Yaskawa INFORM job: MASTER_X2.JBI

/JOB
//NAME MASTER_X2
///FOLDERNAME MASTER_ODWLOK
//POS
///NPOS 131,131,131,0,0,0
///TOOL 0
///POSTYPE PULSE
///PULSE
C00000=-2000,-113621,-91819,0,89172,0
C00001=-2000,-113621,-91819,0,89172,0
C00002=-2032,-101495,-83135,17,53290,-13
C00003=-2000,-48025,-60869,0,102856,0
C00004=-3643,-76224,-106676,-19950,71810,-76872
C00005=-3643,-76224,-106676,-19950,71810,-76872
C00006=-2000,-130321,-133031,0,28968,0
C00007=-2000,-109649,-128472,0,44436,0
C00008=-2000,-75195,-120874,0,70216,0
C00009=-2000,-52226,-115808,0,87402,0
C00010=-2000,-87067,-95572,0,78525,0
C00011=-2000,-87067,-95572,0,78525,0
C00012=-2000,-87067,-95572,0,78525,0
C00013=12667,-135547,-130714,-31270,45596,0
C00014=12667,-135547,-130714,-31270,45596,0
C00015=12667,-135547,-130714,-31270,45596,0
C00016=7337,-135032,-132177,-15524,30149,-37578
C00017=1415,-134459,-133802,1969,12985,-79332
C00018=1415,-134459,-133802,1969,12985,-79332
C00019=15972,-110889,-128286,10965,59905,43045
C00020=-2800,-56338,-97337,367,83074,-232
C00021=-2800,-56338,-97337,367,83074,-232
C00022=-2000,-92772,-84335,0,66375,0
C00023=-2000,-92772,-84335,0,66375,0
C00024=-2000,-92772,-84335,0,66375,0
C00025=-2000,-92772,-84335,0,66375,0
C00026=-2000,-92055,-48789,0,51065,0
C00027=-2000,-92055,-48789,0,51065,0
C00028=-2000,-92055,-48789,0,51065,0
C00029=-2000,-92055,-48789,0,51065,0
C00030=-2348,-136985,-121477,-16,96092,-119
C00031=-2348,-136985,-121477,-16,96092,-119
C00032=-2348,-136985,-121477,-16,96092,-119
C00033=9622,-119744,-117240,-5707,89112,-22022
C00034=39612,-76551,-106625,-19964,71626,-76894
C00035=8691,-94790,-119167,-5108,91578,-19600
C00036=-1903,-101039,-123464,-18,98414,30
C00037=-1903,-101039,-123464,-18,98414,30
C00038=-1903,-101039,-123464,-18,98414,30
C00039=-1903,-101039,-123464,-18,98414,30
C00040=39612,-76551,-106625,-19964,71626,-76894
C00041=39612,-76551,-106625,-19964,71626,-76894
C00042=39612,-76551,-106625,-19964,71626,-76894
C00043=39612,-76551,-106625,-19964,71626,-76894
C00044=39612,-76551,-106625,-19964,71626,-76894
C00045=39612,-76551,-106625,-19964,71626,-76894
C00046=39612,-76551,-106625,-19964,71626,-76894
C00047=39612,-76551,-106625,-19964,71626,-76894
C00048=39612,-76551,-106625,-19964,71626,-76894
C00049=10776,-116726,-133110,-1428,79202,-268
C00050=10776,-116726,-133110,-1428,79202,-268
C00051=10907,-117335,-90652,18762,63715,59495
C00052=10907,-117335,-90652,18762,63715,59495
C00053=10776,-116726,-133110,-1428,79202,-268
C00054=10776,-116726,-133110,-1428,79202,-268
C00055=10907,-117335,-90652,18762,63715,59495
C00056=-2286,-107682,-96534,81,71711,-101
C00057=-2286,-107682,-96534,81,71711,-101
C00058=-2286,-107682,-96534,81,71711,-101
C00059=-2000,-113393,-91320,0,88983,0
C00060=-2000,-113393,-91320,0,88983,0
C00061=-2000,-113393,-91320,0,88983,0
C00062=-2000,-113393,-91320,0,88983,0
C00063=-2000,-113393,-91320,0,88983,0
C00064=39612,-76551,-106625,-19964,71626,-76894
C00065=39612,-76551,-106625,-19964,71626,-76894
C00066=39612,-76551,-106625,-19964,71626,-76894
C00067=39612,-76551,-106625,-19964,71626,-76894
C00068=39612,-76551,-106625,-19964,71626,-76894
C00069=39612,-76551,-106625,-19964,71626,-76894
C00070=-15532,205449,169164,0,-1122,-37
C00071=2435,135546,115697,-1555,71481,-4054
C00072=2435,135546,115697,-1555,71481,-4054
C00073=-5072,204191,173913,2520,2133,2072
C00074=-5072,204191,173913,2520,52116,2072
C00075=-3643,-76224,-106676,-19950,71810,-76872
C00076=-1588,-95931,-85547,536,91020,79
C00077=-1588,-95931,-85547,536,91020,79
C00078=-2000,-138093,-117084,0,0,0
C00079=-3643,-76224,-106676,-19950,71810,-76872
C00080=-2000,-138093,-117084,0,0,0
C00081=-2000,-138093,-117084,0,0,0
C00082=-1941,-102693,-129564,-10,101994,18
C00083=-3643,-76224,-106676,-19950,71810,-76872
C00084=-1074,-84890,-111921,-820,92639,133
C00085=-1074,-84890,-111921,-820,92639,133
C00086=-1999,-107637,-123410,0,80759,-1
C00087=-3643,-76224,-106676,-19950,71810,-76872
C00088=-2000,17994,-60377,0,102988,0
C00089=-2000,-95440,-72516,0,38121,0
C00090=-1074,-84890,-111921,-820,92639,133
C00091=-3643,-76224,-106676,-19950,71810,-76872
C00092=-421,-73083,-90384,286,80877,488
C00093=-421,-73083,-90384,286,80877,488
C00094=-2000,-112988,-119327,0,83158,0
C00095=-3643,-76224,-106676,-19950,71810,-76872
C00096=-2000,-112988,-119327,0,83158,0
C00097=-2000,-112988,-119327,0,83158,0
C00098=-2000,-112988,-119327,0,83158,0
C00099=-2000,-112988,-119327,0,83158,0
C00100=-2082,-130750,-111396,32,62200,-31
C00101=-3643,-76224,-106676,-19950,71810,-76872
C00102=-2082,-130750,-111396,32,62200,-31
C00103=-2082,-130750,-111396,32,62200,-31
C00104=-1579,-114561,-88072,-141,60969,160
C00105=-1579,-114561,-88072,-141,60969,160
C00106=-1579,-114561,-88072,-141,60969,160
C00107=-3643,-76224,-106676,-19950,71810,-76872
C00108=137109,-187493,-133090,-6705,82774,76786
C00109=-3643,-76224,-106676,-19950,71810,-76872
C00110=-1579,-114561,-88072,-141,60969,160
C00111=-2027,-78555,-65913,-1,89981,-9
C00112=-3643,-76224,-106676,-19950,71810,-76872
C00113=-2027,-78555,-65913,-1,89981,-9
C00114=-2027,-78555,-65913,-1,89981,-9
C00115=-3322,-122452,-100913,73,83322,-449
C00116=-3643,-76224,-106676,-19950,71810,-76872
C00117=-3322,-122452,-100913,73,83322,-449
C00118=-3322,-122452,-100913,73,83322,-449
C00119=-3322,-122452,-100913,73,83322,-449
C00120=-3322,-122452,-100913,73,83322,-449
C00121=-3322,-122452,-100913,73,83322,-449
C00122=-2847,-120416,-115970,194,80716,-285
C00123=-2000,-115920,-83969,0,54247,0
C00124=-2000,-115920,-83969,0,54247,0
C00125=-3271,-119374,-120746,350,28955,-423
C00126=-3271,-119374,-120746,350,28955,-423
C00127=-3270,-119374,-120745,350,28960,-423
C00128=-3270,-119374,-120745,350,28960,-423
C00129=-3271,-119374,-120746,350,28955,-423
C00130=-2000,-115588,-91819,0,89172,0
BC00000=87173,519039,860034
BC00001=87173,500620,1075193
BC00002=1577,523905,302382
BC00003=118448,523905,678960
BC00004=199448,515539,1075137
BC00005=199448,515539,1075137
BC00006=200118,491577,1075193
BC00007=160304,500134,1054011
BC00008=93948,514396,1018707
BC00009=49710,523905,995172
BC00010=66564,515818,1075139
BC00011=66564,515818,1075139
BC00012=66564,515818,1075139
BC00013=78377,519142,1075139
BC00014=78377,519142,1075139
BC00015=78377,519142,1075139
BC00016=64373,510676,1075139
BC00017=48813,501269,1075139
BC00018=48813,501269,1075139
BC00019=21198,517278,1075139
BC00020=194066,523905,1075139
BC00021=194066,523905,1075139
BC00022=244938,523905,1064782
BC00023=244938,523905,1063114
BC00024=244938,523905,804554
BC00025=244938,523905,1062363
BC00026=198867,523905,1060460
BC00027=198867,523905,1063860
BC00028=198867,523905,632202
BC00029=198867,523905,632202
BC00030=133244,518772,1075139
BC00031=133244,518772,1075139
BC00032=133244,518772,1075139
BC00033=179478,517852,1075139
BC00034=295309,515546,1075139
BC00035=207944,518721,1071325
BC00036=178010,519809,1070018
BC00037=178010,519809,1070018
BC00038=178010,519809,1070018
BC00039=178010,519809,1070018
BC00040=295309,515546,1075139
BC00041=295309,515546,1075139
BC00042=295309,515546,1075139
BC00043=295309,515546,1075139
BC00044=295309,515546,1075139
BC00045=295309,515546,1075139
BC00046=295309,515546,1075139
BC00047=295309,515546,1075139
BC00048=295309,515546,1075139
BC00049=165804,522273,1075193
BC00050=165804,522273,1075193
BC00051=165804,522273,534000
BC00052=165804,608579,806934
BC00053=165804,522273,1075193
BC00054=165804,522273,1075193
BC00055=165804,522273,534000
BC00056=84290,518606,1075193
BC00057=84290,518606,1075193
BC00058=84290,518606,1075193
BC00059=87173,523905,1075193
BC00060=87173,523905,1075193
BC00061=87173,523905,1075193
BC00062=87173,523905,1075193
BC00063=87173,523905,1075193
BC00064=295309,515546,1075139
BC00065=295309,515546,1075139
BC00066=295309,515546,1075139
BC00067=295309,515546,1075139
BC00068=295309,515546,1075139
BC00069=295309,515546,1075139
BC00070=1577,514581,1075193
BC00071=23362,568996,1042628
BC00072=23362,568996,1042628
BC00073=21044,590463,17935
BC00074=21044,590463,17935
BC00075=199448,582493,1075137
BC00076=197629,523905,680388
BC00077=197629,523905,680388
BC00078=166704,523889,1057027
BC00079=199448,515539,1075137
BC00080=166704,523889,1057027
BC00081=166704,523889,1057027
BC00082=210602,521349,578617
BC00083=199448,515539,1075137
BC00084=166156,519383,387149
BC00085=166156,519383,1064329
BC00086=108222,519829,1065853
BC00087=199448,515539,1075137
BC00088=32574,515576,986534
BC00089=30845,523905,744523
BC00090=166156,519383,1045384
BC00091=199448,515539,1075137
BC00092=146427,523905,652589
BC00093=146427,523905,652589
BC00094=91885,523905,1075139
BC00095=199448,515539,1075137
BC00096=91885,523905,1075139
BC00097=91885,523905,1075139
BC00098=91885,523905,1075139
BC00099=91885,523905,1075139
BC00100=147852,523905,1075139
BC00101=199448,515539,1075137
BC00102=147852,523905,1075139
BC00103=147852,523905,1075139
BC00104=127037,517515,1075193
BC00105=127037,517515,1075193
BC00106=127037,517515,1075193
BC00107=199448,515539,1075137
BC00108=267017,506351,1057956
BC00109=199448,515539,1075137
BC00110=127037,517515,1075193
BC00111=1577,523905,1063536
BC00112=199448,515539,1075137
BC00113=1577,523905,619430
BC00114=1577,523905,619430
BC00115=87745,523889,1075193
BC00116=199448,515539,1075137
BC00117=87745,523889,1075193
BC00118=87745,523889,1075193
BC00119=87745,523889,1075193
BC00120=87745,523889,1075193
BC00121=87745,523889,1075193
BC00122=780,523905,878730
BC00123=262874,523905,990511
BC00124=262874,523905,990511
BC00125=132367,523905,1075193
BC00126=132367,523905,1075193
BC00127=132367,523905,1075190
BC00128=132367,523905,1075190
BC00129=132367,523905,1075193
BC00130=86218,606896,448189
EC00000=0,-183832
EC00001=0,-183832
EC00002=-798156,-183832
EC00003=-798156,-1296783
EC00004=-798156,-1296783
EC00005=-306282,-1296783
EC00006=798156,-1296783
EC00007=869104,-1018545
EC00008=869104,-462069
EC00009=798156,-183832
EC00010=798156,-1296783
EC00011=266052,-1296783
EC00012=-266052,-183832
EC00013=-798156,-183832
EC00014=-798156,-183832
EC00015=-266052,-183832
EC00016=-266052,-740307
EC00017=-266052,-1296783
EC00018=-798156,-1296783
EC00019=-798156,-1296783
EC00020=798156,-183832
EC00021=266052,-183832
EC00022=-266052,-1296783
EC00023=-798156,-1296783
EC00024=-798156,-1296783
EC00025=-266052,-1296783
EC00026=5855,-183832
EC00027=-798156,-183832
EC00028=-798156,-183832
EC00029=-266052,-183832
EC00030=443420,372643
EC00031=798156,372643
EC00032=266052,372643
EC00033=-240191,-131321
EC00034=-1507629,-183832
EC00035=-1445784,372643
EC00036=-1330261,372643
EC00037=-1330261,372643
EC00038=-1596313,372643
EC00039=-1507629,-183832
EC00040=1507629,-183832
EC00041=1596313,372643
EC00042=1463287,372643
EC00043=1463287,372643
EC00044=1463287,372643
EC00045=1463287,372643
EC00046=1596313,372643
EC00047=1596313,-183832
EC00048=266052,-183832
EC00049=-266052,-1296783
EC00050=-798156,-1296783
EC00051=-798156,-1296783
EC00052=-266052,-1296783
EC00053=-266052,-183832
EC00054=-798156,-183832
EC00055=-798156,-183832
EC00056=-798156,-183832
EC00057=-798156,-183832
EC00058=-266052,-183832
EC00059=-266052,-1296783
EC00060=-798156,-1296783
EC00061=-798156,-1296783
EC00062=-266052,-1296783
EC00063=266052,-183832
EC00064=1507629,-183832
EC00065=1596313,372643
EC00066=1463287,372643
EC00067=1463287,372643
EC00068=1596313,372643
EC00069=1507629,-183832
EC00070=266052,-183832
EC00071=-2992,-740304
EC00072=1108548,-740304
EC00073=1108551,-740307
EC00074=1108551,-740307
EC00075=-798155,-740307
EC00076=-798156,-740307
EC00077=-266052,-740307
EC00078=-266052,372643
EC00079=-798156,372643
EC00080=-798156,372643
EC00081=-266052,372643
EC00082=-266052,-183832
EC00083=-798156,-183832
EC00084=-798156,-183832
EC00085=-266052,-183832
EC00086=266050,-1296783
EC00087=798156,-1296783
EC00088=798156,-183832
EC00089=266052,-183832
EC00090=-266052,-1296783
EC00091=-798156,-1296783
EC00092=-798156,-1296783
EC00093=-1596313,-1296783
EC00094=-1596313,372643
EC00095=-1330261,372643
EC00096=-1330261,372643
EC00097=-1596313,372643
EC00098=-1507629,-183832
EC00099=-266052,-183832
EC00100=-266052,-740307
EC00101=-780419,-740307
EC00102=-780419,-740307
EC00103=-266052,-740307
EC00104=266052,-183832
EC00105=798156,-183832
EC00106=1585256,-183832
EC00107=1527674,-741132
EC00108=1488721,-182878
EC00109=798156,-183832
EC00110=-266052,-183832
EC00111=-266052,-740307
EC00112=-798154,-740306
EC00113=-798156,-740307
EC00114=-266052,-740307
EC00115=-266052,-1296783
EC00116=-798156,-1296783
EC00117=-798156,-1296783
EC00118=-266052,-1296783
EC00119=-266052,-183832
EC00120=-798156,-183832
EC00121=-798156,-183832
EC00122=-1596313,-183832
EC00123=-1596313,372643
EC00124=-1596313,-183832
EC00125=-266052,-183832
EC00126=-266052,-740307
EC00127=77843,371283
EC00128=77843,371283
EC00129=0,-183832
EC00130=0,-183832
//INST
///DATE 2024/12/18 17:27
///ATTR SC,RW
///GROUP1 RB1,BS1
///GROUP2 ST1
NOP
WAIT IG#(285)=255
CLEAR B060 1
'MASTER
SETTM TM000 TRESET
SETTM TM000 TSTART
COMM DOUT OT#(1433) ON
DOUT OT#(1437) ON
MOVJ C00000 BC00000 VJ=100.00  +MOVJ EC00000 VJ=100.00
MOVJ C00001 BC00001 VJ=100.00  +MOVJ EC00001 VJ=100.00
CALL JOB:CLEAN-R1_KM_NEW
MOVJ C00002 BC00002 VJ=100.00  +MOVJ EC00002 VJ=100.00
CALL JOB:X2_99(90,0)
MOVJ C00003 BC00003 VJ=100.00  +MOVJ EC00003 VJ=100.00
'
'
MOVJ C00004 BC00004 VJ=100.00  +MOVJ EC00004 VJ=100.00
MOVJ C00005 BC00005 VJ=100.00  +MOVJ EC00005 VJ=100.00
CALL JOB:CLEAN-R1_KM_NEW
CALL JOB:X2_R2_O242(-90,180)NEW
MOVJ C00006 BC00006 VJ=100.00  +MOVJ EC00006 VJ=100.00
'
MOVJ C00007 BC00007 VJ=100.00  +MOVJ EC00007 VJ=100.00
MOVJ C00008 BC00008 VJ=100.00  +MOVJ EC00008 VJ=100.00
'
SFTOF3D
MOVJ C00009 BC00009 VJ=100.00  +MOVJ EC00009 VJ=100.00
CALL JOB:CLEAN-R1_KM_NEW
CALL JOB:X2_6-7(-90,0)
MOVJ C00010 BC00010 VJ=100.00  +MOVJ EC00010 VJ=100.00
'
MOVJ C00011 BC00011 VJ=100.00  +MOVJ EC00011 VJ=100.00
MOVJ C00012 BC00012 VJ=100.00  +MOVJ EC00012 VJ=100.00
'
MOVJ C00013 BC00013 VJ=100.00  +MOVJ EC00013 VJ=100.00
CALL JOB:X2_8A-21A(90,0)
MOVJ C00014 BC00014 VJ=100.00  +MOVJ EC00014 VJ=100.00
'
MOVJ C00015 BC00015 VJ=100.00  +MOVJ EC00015 VJ=100.00
MOVJ C00016 BC00016 VJ=100.00  +MOVJ EC00016 VJ=100.00
MOVJ C00017 BC00017 VJ=100.00  +MOVJ EC00017 VJ=100.00
'
MOVJ C00018 BC00018 VJ=100.00  +MOVJ EC00018 VJ=100.00
CALL JOB:CLEAN-R1_KM_NEW
CALL JOB:X2_8B-21B(90,180)
MOVJ C00019 BC00019 VJ=100.00  +MOVJ EC00019 VJ=100.00
CALL JOB:CLEAN-R1_KM_NEW
'
'
CALL JOB:X2_22-23(-90,180)
MOVJ C00020 BC00020 VJ=100.00  +MOVJ EC00020 VJ=100.00
'
MOVJ C00021 BC00021 VJ=100.00  +MOVJ EC00021 VJ=100.00
MOVJ C00022 BC00022 VJ=100.00  +MOVJ EC00022 VJ=100.00
'
MOVJ C00023 BC00023 VJ=100.00  +MOVJ EC00023 VJ=100.00
CALL JOB:CLEAN-R1_KM_NEW
CALL JOB:X2_24A(90,180)
MOVJ C00024 BC00024 VJ=100.00  +MOVJ EC00024 VJ=100.00
'
MOVJ C00025 BC00025 VJ=100.00  +MOVJ EC00025 VJ=100.00
MOVJ C00026 BC00026 VJ=100.00  +MOVJ EC00026 VJ=100.00
'
MOVJ C00027 BC00027 VJ=100.00  +MOVJ EC00027 VJ=100.00
CALL JOB:CLEAN-R1_KM_NEW
CALL JOB:X2_24B(90,0)
MOVJ C00028 BC00028 VJ=100.00  +MOVJ EC00028 VJ=100.00
'
MOVJ C00029 BC00029 VJ=100.00  +MOVJ EC00029 VJ=100.00
'
MOVJ C00030 BC00030 VJ=100.00  +MOVJ EC00030 VJ=100.00
CALL JOB:CLEAN-R1_KM_NEW
CALL JOB:X2_27-28(-50,-90)
MOVJ C00031 BC00031 VJ=100.00  +MOVJ EC00031 VJ=100.00
'NOWY PRZEJAZD
'
MOVJ C00032 BC00032 VJ=100.00  +MOVJ EC00032 VJ=100.00
MOVJ C00033 BC00033 VJ=100.00  +MOVJ EC00033 VJ=100.00
MOVJ C00034 BC00034 VJ=100.00  +MOVJ EC00034 VJ=100.00
MOVJ C00035 BC00035 VJ=100.00  +MOVJ EC00035 VJ=100.00
'
MOVJ C00036 BC00036 VJ=100.00  +MOVJ EC00036 VJ=100.00
CALL JOB:X2_7,2(150,-90)
MOVJ C00037 BC00037 VJ=100.00  +MOVJ EC00037 VJ=100.00
'
MOVJ C00038 BC00038 VJ=100.00  +MOVJ EC00038 VJ=100.00
MOVJ C00039 BC00039 VJ=100.00  +MOVJ EC00039 VJ=100.00
MOVJ C00040 BC00040 VJ=100.00  +MOVJ EC00040 VJ=100.00
MOVJ C00041 BC00041 VJ=100.00  +MOVJ EC00041 VJ=100.00
'
MOVJ C00042 BC00042 VJ=100.00  +MOVJ EC00042 VJ=100.00
CALL JOB:CLEAN-R1_KM_NEW
CALL JOB:X2_7,1(-165,-90)0
MOVJ C00043 BC00043 VJ=100.00  +MOVJ EC00043 VJ=100.00
'
'
MOVJ C00044 BC00044 VJ=100.00  +MOVJ EC00044 VJ=100.00
CALL JOB:CLEAN-R1_KM_NEW
CALL JOB:X2_34(P)(-165,-90)
MOVJ C00045 BC00045 VJ=100.00  +MOVJ EC00045 VJ=100.00
'
MOVJ C00046 BC00046 VJ=100.00  +MOVJ EC00046 VJ=100.00
MOVJ C00047 BC00047 VJ=100.00  +MOVJ EC00047 VJ=100.00
MOVJ C00048 BC00048 VJ=100.00  +MOVJ EC00048 VJ=100.00
MOVJ C00049 BC00049 VJ=100.00  +MOVJ EC00049 VJ=100.00
'
MOVJ C00050 BC00050 VJ=100.00  +MOVJ EC00050 VJ=100.00
CALL JOB:CLEAN-R1_KM_NEW
CALL JOB:X2_38-47,64(1)(90,180)
MOVJ C00051 BC00051 VJ=100.00  +MOVJ EC00051 VJ=100.00
'
MOVJ C00052 BC00052 VJ=100.00  +MOVJ EC00052 VJ=100.00
MOVJ C00053 BC00053 VJ=100.00  +MOVJ EC00053 VJ=100.00
'
MOVJ C00054 BC00054 VJ=100.00  +MOVJ EC00054 VJ=100.00
CALL JOB:CLEAN-R1_KM_NEW
CALL JOB:X2_38-47,64(2)(90,0)
MOVJ C00055 BC00055 VJ=100.00  +MOVJ EC00055 VJ=100.00
'
'
MOVJ C00056 BC00056 VJ=100.00  +MOVJ EC00056 VJ=100.00
CALL JOB:CLEAN-R1_KM_NEW
CALL JOB:X2_50&56A(90,0)
MOVJ C00057 BC00057 VJ=100.00  +MOVJ EC00057 VJ=100.00
'
MOVJ C00058 BC00058 VJ=100.00  +MOVJ EC00058 VJ=100.00
MOVJ C00059 BC00059 VJ=100.00  +MOVJ EC00059 VJ=100.00
'
MOVJ C00060 BC00060 VJ=100.00  +MOVJ EC00060 VJ=100.00
CALL JOB:CLEAN-R1_KM_NEW
CALL JOB:X2_50&56B(90_180)
MOVJ C00061 BC00061 VJ=100.00  +MOVJ EC00061 VJ=100.00
'
MOVJ C00062 BC00062 VJ=100.00  +MOVJ EC00062 VJ=100.00
MOVJ C00063 BC00063 VJ=100.00  +MOVJ EC00063 VJ=100.00
MOVJ C00064 BC00064 VJ=100.00  +MOVJ EC00064 VJ=100.00
MOVJ C00065 BC00065 VJ=100.00  +MOVJ EC00065 VJ=100.00
'
MOVJ C00066 BC00066 VJ=100.00  +MOVJ EC00066 VJ=100.00
CALL JOB:CLEAN-R1_KM_NEW
CALL JOB:X2_51(P)(-165,-90)
MOVJ C00067 BC00067 VJ=100.00  +MOVJ EC00067 VJ=100.00
'
MOVJ C00068 BC00068 VJ=100.00  +MOVJ EC00068 VJ=100.00
MOVJ C00069 BC00069 VJ=100.00  +MOVJ EC00069 VJ=100.00
MOVJ C00070 BC00070 VJ=100.00  +MOVJ EC00070 VJ=100.00
'
MOVJ C00071 BC00071 VJ=15.00  +MOVJ EC00071 VJ=15.00
MOVJ C00072 BC00072 VJ=15.00  +MOVJ EC00072 VJ=15.00
CALL JOB:X2_100(P)(125,-90)
'
'
MOVJ C00073 BC00073 VJ=100.00  +MOVJ EC00073 VJ=100.00
MOVJ C00074 BC00074 VJ=100.00  +MOVJ EC00074 VJ=100.00
PAUSE
'UWAGA!!!!!!!!
'WYMIANA KONCOWKI PRADOWEJ
CALL JOB:CLEAN-R1_KM_NEW
CALL JOB:X2_101(P)NEWKM
'
'
MOVJ C00075 BC00075 VJ=100.00  +MOVJ EC00075 VJ=100.00
CALL JOB:CLEAN-R1_KM_NEW
CALL JOB:X2_54(90,90)
MOVJ C00076 BC00076 VJ=100.00  +MOVJ EC00076 VJ=100.00
'
MOVJ C00077 BC00077 VJ=100.00  +MOVJ EC00077 VJ=100.00
MOVJ C00078 BC00078 VJ=100.00  +MOVJ EC00078 VJ=100.00
'
MOVJ C00079 BC00079 VJ=100.00  +MOVJ EC00079 VJ=100.00
CALL JOB:CLEAN-R1_KM_NEW
CALL JOB:X2_102(P)(90,-90)1
MOVJ C00080 BC00080 VJ=100.00  +MOVJ EC00080 VJ=100.00
'
MOVJ C00081 BC00081 VJ=100.00  +MOVJ EC00081 VJ=100.00
MOVJ C00082 BC00082 VJ=100.00  +MOVJ EC00082 VJ=100.00
'
MOVJ C00083 BC00083 VJ=100.00  +MOVJ EC00083 VJ=100.00
CALL JOB:CLEAN-R1_KM_NEW
CALL JOB:X2_57-69(1)(90,0)
MOVJ C00084 BC00084 VJ=100.00  +MOVJ EC00084 VJ=100.00
'
MOVJ C00085 BC00085 VJ=100.00  +MOVJ EC00085 VJ=100.00
MOVJ C00086 BC00086 VJ=100.00  +MOVJ EC00086 VJ=100.00
'
MOVJ C00087 BC00087 VJ=100.00  +MOVJ EC00087 VJ=100.00
CALL JOB:CLEAN-R1_KM_NEW
CALL JOB:X2_29-32(-90,180)
MOVJ C00088 BC00088 VJ=100.00  +MOVJ EC00088 VJ=100.00
'
MOVJ C00089 BC00089 VJ=100.00  +MOVJ EC00089 VJ=100.00
MOVJ C00090 BC00090 VJ=100.00  +MOVJ EC00090 VJ=100.00
'
MOVJ C00091 BC00091 VJ=100.00  +MOVJ EC00091 VJ=100.00
CALL JOB:CLEAN-R1_KM_NEW
CALL JOB:X2_57-69(2)(90,180)
MOVJ C00092 BC00092 VJ=100.00  +MOVJ EC00092 VJ=100.00
'
MOVJ C00093 BC00093 VJ=100.00  +MOVJ EC00093 VJ=100.00
MOVJ C00094 BC00094 VJ=100.00  +MOVJ EC00094 VJ=100.00
'
MOVJ C00095 BC00095 VJ=100.00  +MOVJ EC00095 VJ=100.00
CALL JOB:CLEAN-R1_KM_NEW
CALL JOB:X2_48(150,-90)
MOVJ C00096 BC00096 VJ=100.00  +MOVJ EC00096 VJ=100.00
'
MOVJ C00097 BC00097 VJ=100.00  +MOVJ EC00097 VJ=100.00
MOVJ C00098 BC00098 VJ=100.00  +MOVJ EC00098 VJ=100.00
MOVJ C00099 BC00099 VJ=100.00  +MOVJ EC00099 VJ=100.00
MOVJ C00100 BC00100 VJ=100.00  +MOVJ EC00100 VJ=100.00
'
MOVJ C00101 BC00101 VJ=100.00  +MOVJ EC00101 VJ=100.00
CALL JOB:CLEAN-R1_KM_NEW
CALL JOB:X2_49(88,90)
MOVJ C00102 BC00102 VJ=100.00  +MOVJ EC00102 VJ=100.00
'
MOVJ C00103 BC00103 VJ=100.00  +MOVJ EC00103 VJ=100.00
MOVJ C00104 BC00104 VJ=100.00  +MOVJ EC00104 VJ=100.00
'
MOVJ C00105 BC00105 VJ=100.00  +MOVJ EC00105 VJ=100.00
'NOWY PROGRAM NA SCHODKI
MOVJ C00106 BC00106 VJ=100.00  +MOVJ EC00106 VJ=100.00
MOVJ C00107 BC00107 VJ=100.00  +MOVJ EC00107 VJ=100.00
CALL JOB:CLEAN-R1_KM_NEW
CALL JOB:X2_NOWY2
MOVJ C00108 BC00108 VJ=100.00  +MOVJ EC00108 VJ=100.00
MOVJ C00109 BC00109 VJ=100.00  +MOVJ EC00109 VJ=100.00
CALL JOB:CLEAN-R1_KM_NEW
'PROG DO POP
CALL JOB:X2_34-37(-90,0)
'
MOVJ C00110 BC00110 VJ=100.00  +MOVJ EC00110 VJ=100.00
MOVJ C00111 BC00111 VJ=100.00  +MOVJ EC00111 VJ=100.00
'
MOVJ C00112 BC00112 VJ=100.00  +MOVJ EC00112 VJ=100.00
CALL JOB:CLEAN-R1_KM_NEW
CALL JOB:X2_25(90,90)
MOVJ C00113 BC00113 VJ=100.00  +MOVJ EC00113 VJ=100.00
'
MOVJ C00114 BC00114 VJ=100.00  +MOVJ EC00114 VJ=100.00
MOVJ C00115 BC00115 VJ=100.00  +MOVJ EC00115 VJ=100.00
'
MOVJ C00116 BC00116 VJ=100.00  +MOVJ EC00116 VJ=100.00
CALL JOB:CLEAN-R1_KM_NEW
CALL JOB:X2_55A(90,180)
MOVJ C00117 BC00117 VJ=100.00  +MOVJ EC00117 VJ=100.00
'
MOVJ C00118 BC00118 VJ=100.00  +MOVJ EC00118 VJ=100.00
MOVJ C00119 BC00119 VJ=100.00  +MOVJ EC00119 VJ=100.00
'
MOVJ C00120 BC00120 VJ=100.00  +MOVJ EC00120 VJ=100.00
CALL JOB:CLEAN-R1_KM_NEW
CALL JOB:X2_55B(90,0)
MOVJ C00121 BC00121 VJ=100.00  +MOVJ EC00121 VJ=100.00
'
'
MOVJ C00122 BC00122 VJ=100.00  +MOVJ EC00122 VJ=100.00
CALL JOB:CLEAN-R1_KM_NEW
CALL JOB:X2_104(180,0)
MOVJ C00123 BC00123 VJ=100.00  +MOVJ EC00123 VJ=100.00
'
MOVJ C00124 BC00124 VJ=100.00  +MOVJ EC00124 VJ=100.00
MOVJ C00125 BC00125 VJ=100.00  +MOVJ EC00125 VJ=100.00
'
MOVJ C00126 BC00126 VJ=100.00  +MOVJ EC00126 VJ=100.00
CALL JOB:CLEAN-R1_KM_NEW
CALL JOB:KRIS7NEWX2
'
MOVJ C00127 BC00127 VJ=100.00  +MOVJ EC00127 VJ=100.00
CALL JOB:CLEAN-R1_KM_NEW
CALL JOB:X2_NOWY
COMM DOUT OT#(1433) OFF
DOUT OT#(1437) OFF
MOVJ C00128 BC00128 VJ=100.00  +MOVJ EC00128 VJ=100.00
MOVJ C00129 BC00129 VJ=100.00  +MOVJ EC00129 VJ=100.00
MOVJ C00130 BC00130 VJ=100.00  +MOVJ EC00130 VJ=100.00
SETTM TM000 TSTOP
PAUSE
PAUSE
PAUSE
'
END
